{attribute 'GeneratedUsingTerminal: EL3011-0000-0016'}
{attribute addProperty BoxType "EL3011-0000-0016"}
{attribute addProperty Id "AI_StandardAT %I*AI_Standard_4A3944819WcStateAT %I*WcState_9091E0EB2InfoDataAT %I*InfoData_94A18F5E2"}
{attribute addProperty CRC "2975591319"}
{attribute addProperty Size "13"}
TYPE EL3011_B15BEB97 EXTENDS EtcSlaveTerminalBase_947E5A46 :
STRUCT
	{attribute addProperty Name "AI_Standard"}
	AI_Standard : AI_Standard_4A394481;
	{attribute addProperty Name "WcState"}
	WcState : WcState_9091E0EB;
	{attribute addProperty Name "InfoData"}
	InfoData : InfoData_94A18F5E;
END_STRUCT
END_TYPE

(* stored: Version 1.2.0.0, ProductVersion 3.1.4024.9
   DUT EL3011_B15BEB97: Id {fa860698-23f5-4e53-b86d-c90e97fe0c9d} *)
